
// ===== library types =====

FUNCTION_BLOCK "Tank"   // FB1, LAD
{ S7_Optimized_Access := 'TRUE' }
VERSION : 0.1
   VAR
      Level : Int;
      Tem : Int;
      Pre : Int;
   END_VAR
BEGIN
END_FUNCTION_BLOCK